// Mitsubishi GX Works2 project: main_controller   PLC: FX3U/FX3UC

PROGRAM MAIN
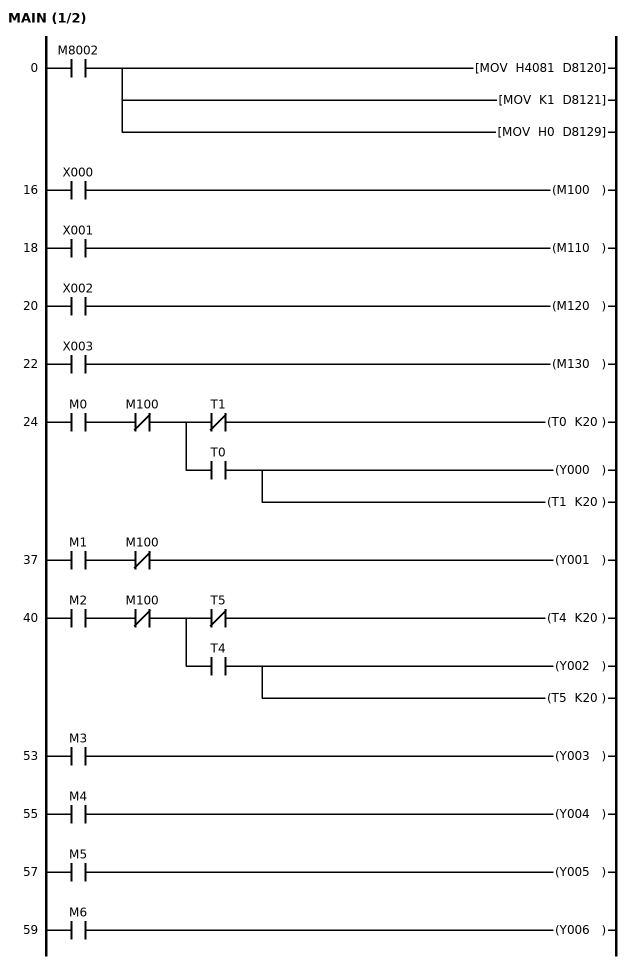
0     LD      M8002
      MOV     H4081 D8120
      MOV     K1 D8121
      MOV     H0 D8129
16    LD      X000
      OUT     M100
18    LD      X001
      OUT     M110
20    LD      X002
      OUT     M120
22    LD      X003
      OUT     M130
24    LD      M0
      ANI     M100
      MPS
      ANI     T1
      OUT     T0 K20
      MPP
      AND     T0
      OUT     Y000
      OUT     T1 K20
37    LD      M1
      ANI     M100
      OUT     Y001
40    LD      M2
      ANI     M100
      MPS
      ANI     T5
      OUT     T4 K20
      MPP
      AND     T4
      OUT     Y002
      OUT     T5 K20
53    LD      M3
      OUT     Y003
55    LD      M4
      OUT     Y004
57    LD      M5
      OUT     Y005
59    LD      M6
      OUT     Y006
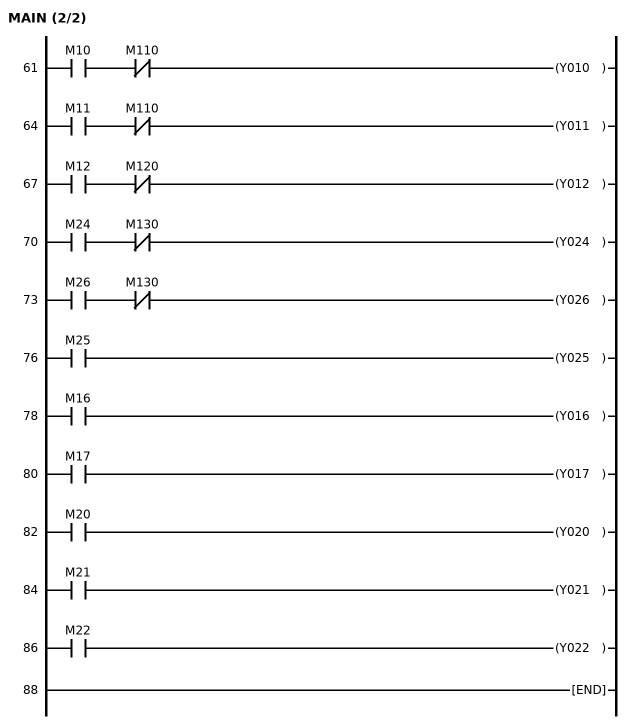
61    LD      M10
      ANI     M110
      OUT     Y010
64    LD      M11
      ANI     M110
      OUT     Y011
67    LD      M12
      ANI     M120
      OUT     Y012
70    LD      M24
      ANI     M130
      OUT     Y024
73    LD      M26
      ANI     M130
      OUT     Y026
76    LD      M25
      OUT     Y025
78    LD      M16
      OUT     Y016
80    LD      M17
      OUT     Y017
82    LD      M20
      OUT     Y020
84    LD      M21
      OUT     Y021
86    LD      M22
      OUT     Y022
88    END
END_PROGRAM
